// TIA Portal V19 export
DATA_BLOCK "DB_Optimierung_HCA"   // DB170
{ S7_Optimized_Access := 'TRUE' }
// stored: AutoNumber false, MemoryReserve 100
   VAR
      Restzeit_Kurz_Links { ExternalWritable := 'False'} : DInt;
      Restzeit_Kurz_Rechts { ExternalWritable := 'False'} : DInt;
      Restzeit_Lang { ExternalWritable := 'False'} : DInt;
      Restzeit_Gross_Links { ExternalWritable := 'False'} : DInt;
      Restzeit_Gross_Rechts { ExternalWritable := 'False'} : DInt;
      Restzeit { ExternalAccessible := 'False'; ExternalVisible := 'False'; ExternalWritable := 'False'} : Array[1..18] of DInt;
   END_VAR
BEGIN
END_DATA_BLOCK
